// Mitsubishi GX Works2 project: ex2 final   PLC: FX3G
// ex2

// global labels: Global1
VAR_GLOBAL
  start_sys AT X007 : BOOL;
  emergency AT X005 : BOOL;
  led_start AT Y007 : BOOL;
  lack_material AT M0 : BOOL;
  lemon_input AT D1100 : REAL;
  lemon_amount AT D1110 : REAL;
  petel_input AT D1120 : REAL;
  petel_amount AT D1130 : REAL;
  stable_input AT D1140 : REAL;
  stable_amount AT D1150 : REAL;
  bear_input AT D1160 : REAL;
  bear_amount AT D1170 : REAL;
  start_flavor AT X001 : BOOL;
  per_400 AT E400 : REAL;
  pinuk_min AT E6 : REAL;
  pinuk_selected AT M1 : BOOL;
  regular_max AT E5 : REAL;
  regular_selected AT M2 : BOOL;
  lemon_min_pinuk AT E665 : REAL;
  check_lemon_pinuk AT M10 : BOOL;
  check_petel_pinuk AT M30 : BOOL;
  petel_min_pinuk AT E385 : REAL;
  stable_min_pinuk AT E210 : REAL;
  check_stable_pinuk AT M50 : BOOL;
  check_bear_pinuk AT M70 : BOOL;
  bear_min_pinuk AT E70 : REAL;
  can_pinuk AT M3 : BOOL;
  check_lemon_reg AT M11 : BOOL;
  lemon_min_reg AT E455 : REAL;
  check_petel_reg AT M31 : BOOL;
  petel_min_reg AT E280 : REAL;
  check_stable_reg AT M51 : BOOL;
  stable_min_reg AT E105 : REAL;
  bear_min_reg AT E28 : REAL;
  check_bear_reg AT M71 : BOOL;
  can_reg AT M4 : BOOL;
  flavor_timer AT TC1 : BOOL;
  done_flavor AT K50 : INT;
  flavor_mix AT TS1 : BOOL;
  flavor_process AT Y000 : BOOL;
  save_analog_input1 AT D7000 : REAL;
  analog_input1 AT D8280 : INT;
  cooling_done AT M7 : BOOL;
  start_blinking AT M8 : BOOL;
  help_blinker AT M9 : BOOL;
  blinkY5 AT TC2 : BOOL;
  blink_time AT K5 : INT;
  blink1 AT TS2 : BOOL;
  lightY5 AT Y005 : BOOL;
  blinkY6 AT TC3 : BOOL;
  blink2 AT TS3 : BOOL;
  lightY6 AT Y006 : BOOL;
  mix_pinuk AT TS4 : BOOL;
  mix_reg AT TS5 : BOOL;
  done_mix_pinuk AT K50 : INT;
  done_mix_reg AT K30 : INT;
  mix_pinuk_timer AT TC4 : BOOL;
  mix_reg_timer AT TC5 : BOOL;
  pinuk_max AT E10 : REAL;
  regular_min AT E0 : REAL;
  finish_ice_making AT M5 : BOOL;
  start_cool AT X002 : BOOL;
  cool_timer AT TS6 : BOOL;
END_VAR
VAR_GLOBAL CONSTANT
  t_value : INT := 80;
END_VAR
VAR_GLOBAL
  cool_run AT TC6 : BOOL;
  cool_indicator AT Y002 : BOOL;
  finish_cool AT X003 : BOOL;
  start_packege AT X004 : BOOL;
  unit_pack AT X000 : BOOL;
  units_num AT CC1 : BOOL;
END_VAR
VAR_GLOBAL CONSTANT
  const7 : INT := 7;
END_VAR
VAR_GLOBAL
  packege_done AT CS1 : BOOL;
  packege_in_process AT Y004 : BOOL;
  packege_inventory AT D6000 : INT;
END_VAR
VAR_GLOBAL CONSTANT
  const1 : INT := 1;
  const10 : INT := 10;
  K_40 : INT := 40;
END_VAR
VAR_GLOBAL
  analog_output AT D8282 : INT;
  cool_lemon AT D7100 : REAL;
  cool_petel AT D7500 : REAL;
  mix_flavor AT D7400 : REAL;
  mix_with_bear AT D7600 : REAL;
  petel_ice_reg AT E350 : REAL;
  lemon_ice_reg AT E490 : REAL;
  petel_ice_pinuk AT E560 : REAL;
  lemon_ice_pinuk AT E700 : REAL;
END_VAR
VAR_GLOBAL CONSTANT
  bear_reg : REAL := E28;
  bear_pinuk : REAL := E70;
END_VAR
VAR_GLOBAL
  packege_indicator AT M6 : BOOL;
END_VAR

// task Task_01 (event TRUE, interval 0, priority 31): POU_01

PROGRAM POU_01
(* structured ladder/FBD written out as ST: instructions are called as NAME(EN, inputs, outputs); _pN, _eN, _tN stand for wires *)
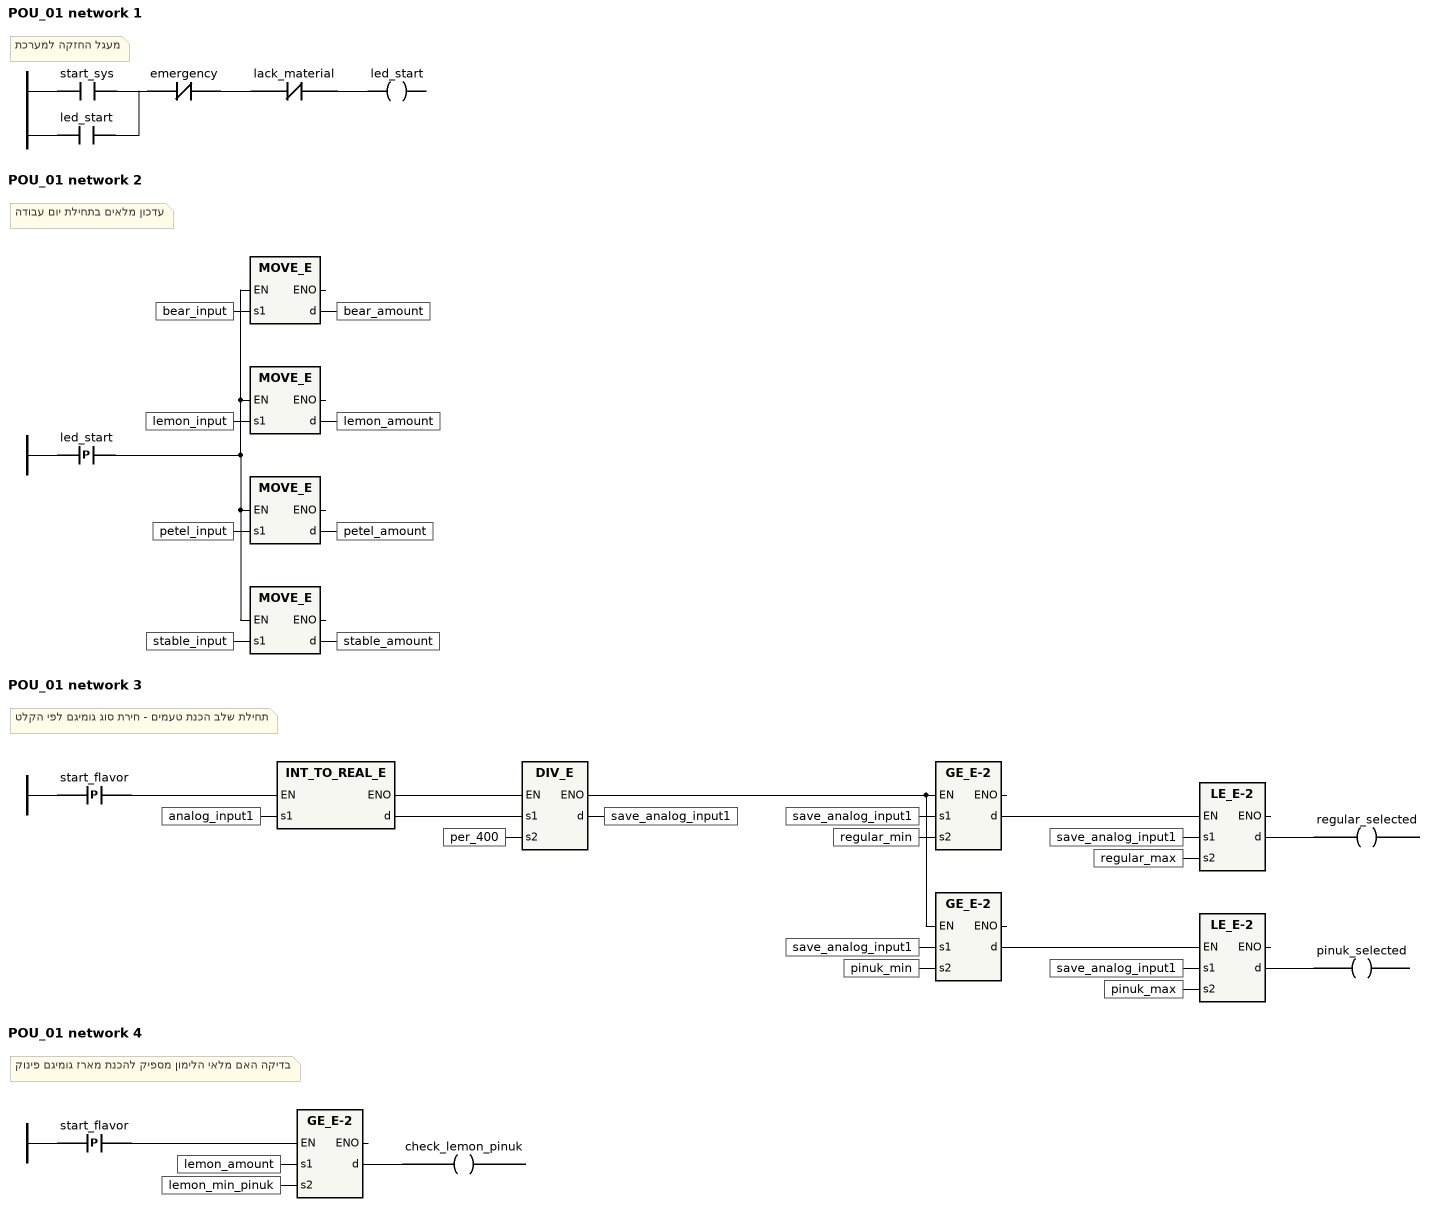
(* network 1 *)
(* מעגל החזקה למערכת *)
led_start := ((start_sys OR led_start) AND NOT emergency) AND NOT lack_material;
(* network 2 *)
(* עדכון מלאים בתחילת יום עבודה *)
_p1 := LDP(TRUE, led_start);
MOVE_E(_p1, bear_input, bear_amount);
MOVE_E(_p1, lemon_input, lemon_amount);
MOVE_E(_p1, petel_input, petel_amount);
MOVE_E(_p1, stable_input, stable_amount);
(* network 3 *)
(* תחילת שלב הכנת טעמים - חירת סוג גומיגם לפי הקלט *)
_e2 := INT_TO_REAL_E(LDP(TRUE, start_flavor), analog_input1, _t1);
_e3 := DIV_E(_e2, _t1, per_400, save_analog_input1);
GE_E(_e3, save_analog_input1, regular_min, _t4);
LE_E(_t4, save_analog_input1, regular_max, _t5);
regular_selected := _t5;
GE_E(_e3, save_analog_input1, pinuk_min, _t6);
LE_E(_t6, save_analog_input1, pinuk_max, _t7);
pinuk_selected := _t7;
(* network 4 *)
(* בדיקה האם מלאי הלימון מספיק להכנת מארז גומיגם פינוק *)
GE_E(LDP(TRUE, start_flavor), lemon_amount, lemon_min_pinuk, _t1);
check_lemon_pinuk := _t1;
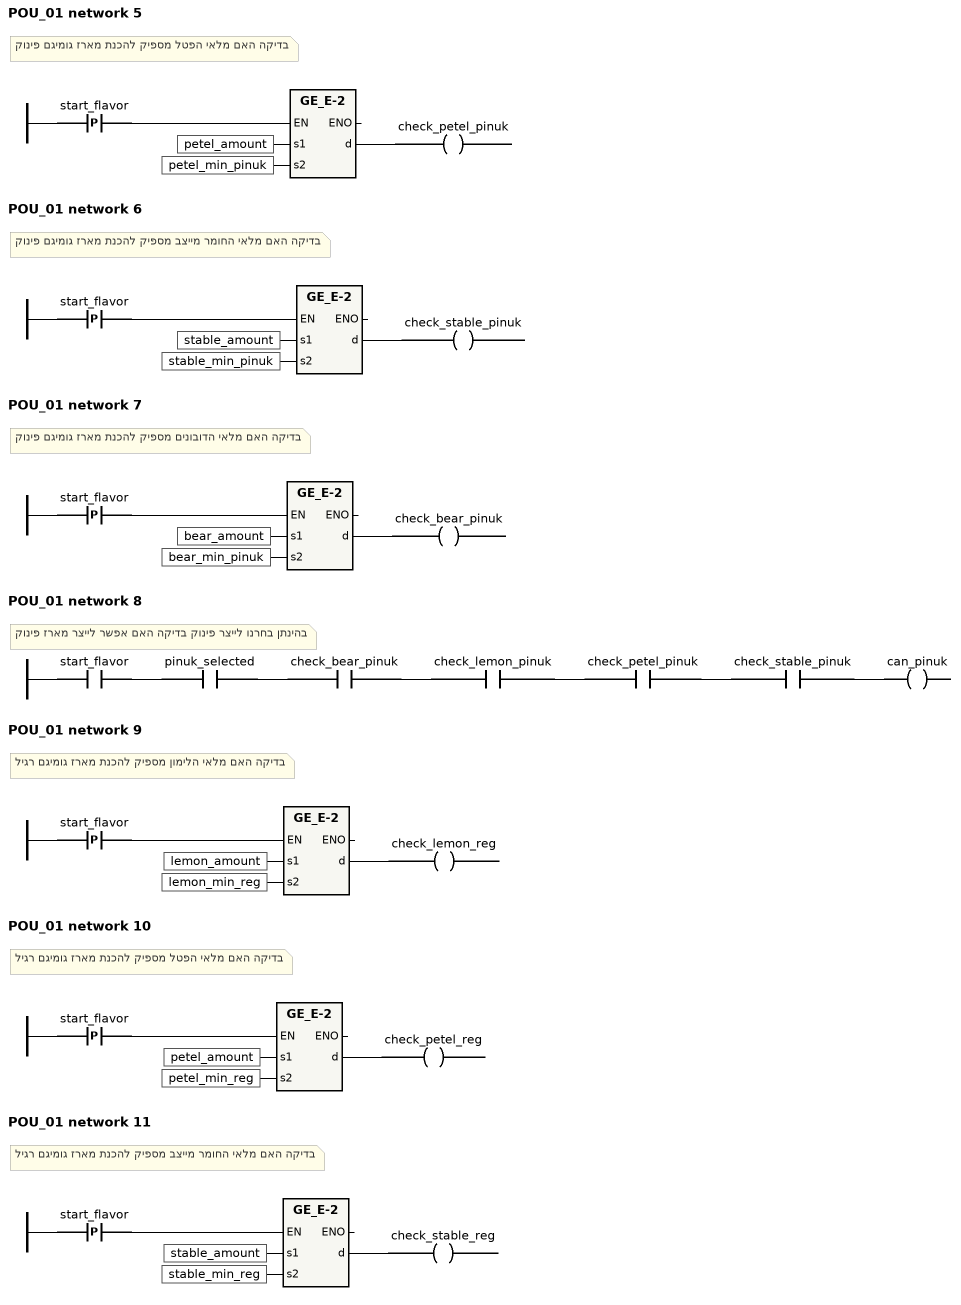
(* network 5 *)
(* בדיקה האם מלאי הפטל מספיק להכנת מארז גומיגם פינוק *)
GE_E(LDP(TRUE, start_flavor), petel_amount, petel_min_pinuk, _t1);
check_petel_pinuk := _t1;
(* network 6 *)
(* בדיקה האם מלאי החומר מייצב מספיק להכנת מארז גומיגם פינוק *)
GE_E(LDP(TRUE, start_flavor), stable_amount, stable_min_pinuk, _t1);
check_stable_pinuk := _t1;
(* network 7 *)
(* בדיקה האם מלאי הדובונים מספיק להכנת מארז גומיגם פינוק *)
GE_E(LDP(TRUE, start_flavor), bear_amount, bear_min_pinuk, _t1);
check_bear_pinuk := _t1;
(* network 8 *)
(* בהינתן בחרנו לייצר פינוק בדיקה האם אפשר לייצר מארז פינוק *)
can_pinuk := start_flavor AND pinuk_selected AND check_bear_pinuk AND check_lemon_pinuk AND check_petel_pinuk AND check_stable_pinuk;
(* network 9 *)
(* בדיקה האם מלאי הלימון מספיק להכנת מארז גומיגם רגיל *)
GE_E(LDP(TRUE, start_flavor), lemon_amount, lemon_min_reg, _t1);
check_lemon_reg := _t1;
(* network 10 *)
(* בדיקה האם מלאי הפטל מספיק להכנת מארז גומיגם רגיל *)
GE_E(LDP(TRUE, start_flavor), petel_amount, petel_min_reg, _t1);
check_petel_reg := _t1;
(* network 11 *)
(* בדיקה האם מלאי החומר מייצב מספיק להכנת מארז גומיגם רגיל *)
GE_E(LDP(TRUE, start_flavor), stable_amount, stable_min_reg, _t1);
check_stable_reg := _t1;
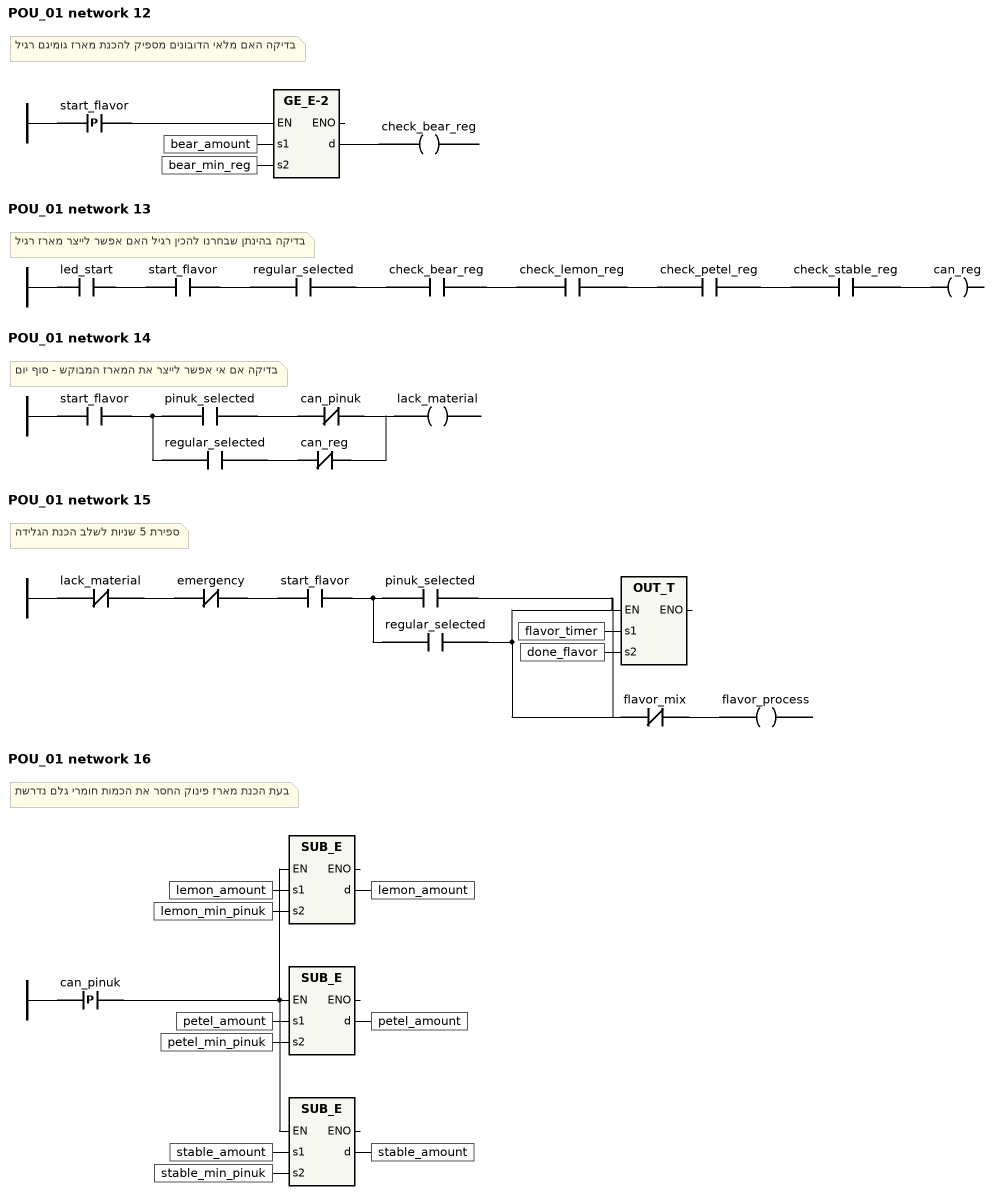
(* network 12 *)
(* בדיקה האם מלאי הדובונים מספיק להכנת מארז גומיגם רגיל *)
GE_E(LDP(TRUE, start_flavor), bear_amount, bear_min_reg, _t1);
check_bear_reg := _t1;
(* network 13 *)
(* בדיקה בהינתן שבחרנו להכין רגיל האם אפשר לייצר מארז רגיל *)
can_reg := led_start AND start_flavor AND regular_selected AND check_bear_reg AND check_lemon_reg AND check_petel_reg AND check_stable_reg;
(* network 14 *)
(* בדיקה אם אי אפשר לייצר את המארז המבוקש - סוף יום *)
lack_material := (start_flavor AND pinuk_selected AND NOT can_pinuk) OR (start_flavor AND regular_selected AND NOT can_reg);
(* network 15 *)
(* ספירת 5 שניות לשלב הכנת הגלידה *)
_p1 := NOT lack_material AND NOT emergency AND start_flavor;
_p2 := (_p1 AND pinuk_selected) OR (_p1 AND regular_selected);
flavor_process := _p2 AND NOT flavor_mix;
OUT_T(_p2, flavor_timer, done_flavor);
(* network 16 *)
(* בעת הכנת מארז פינוק החסר את הכמות חומרי גלם נדרשת *)
_p1 := LDP(TRUE, can_pinuk);
SUB_E(_p1, lemon_amount, lemon_min_pinuk, lemon_amount);
SUB_E(_p1, petel_amount, petel_min_pinuk, petel_amount);
SUB_E(_p1, stable_amount, stable_min_pinuk, stable_amount);
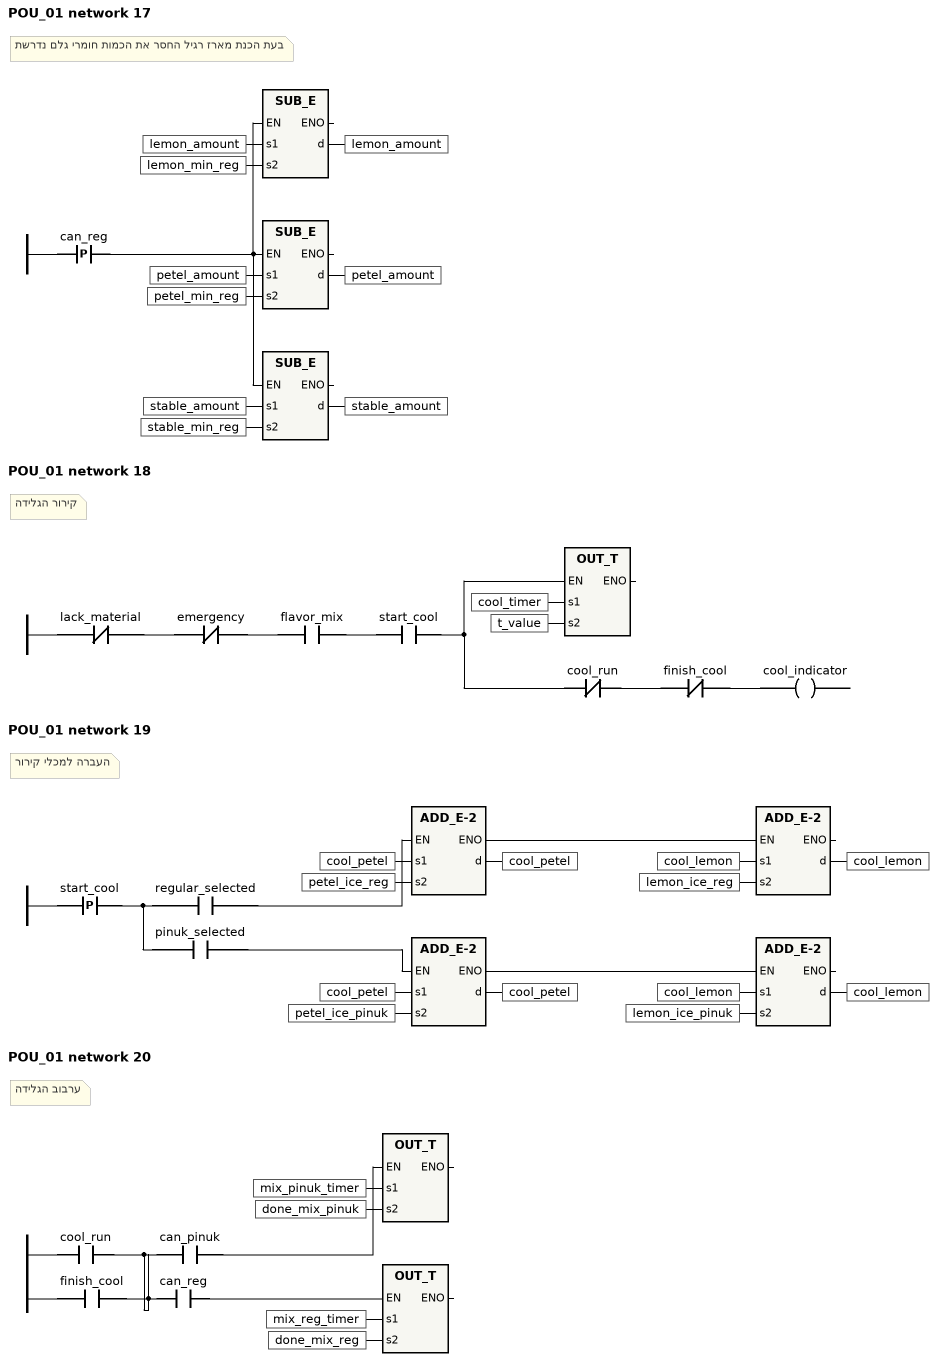
(* network 17 *)
(* בעת הכנת מארז רגיל החסר את הכמות חומרי גלם נדרשת *)
_p1 := LDP(TRUE, can_reg);
SUB_E(_p1, lemon_amount, lemon_min_reg, lemon_amount);
SUB_E(_p1, petel_amount, petel_min_reg, petel_amount);
SUB_E(_p1, stable_amount, stable_min_reg, stable_amount);
(* network 18 *)
(* קירור הגלידה *)
_p1 := NOT lack_material AND NOT emergency AND flavor_mix AND start_cool;
OUT_T(_p1, cool_timer, t_value);
cool_indicator := _p1 AND NOT cool_run AND NOT finish_cool;
(* network 19 *)
(* העברה למכלי קירור *)
_p1 := LDP(TRUE, start_cool);
_e2 := ADD_E(_p1 AND regular_selected, cool_petel, petel_ice_reg, cool_petel);
ADD_E(_e2, cool_lemon, lemon_ice_reg, cool_lemon);
_e3 := ADD_E(_p1 AND pinuk_selected, cool_petel, petel_ice_pinuk, cool_petel);
ADD_E(_e3, cool_lemon, lemon_ice_pinuk, cool_lemon);
(* network 20 *)
(* ערבוב הגלידה *)
_p1 := cool_run OR finish_cool;
OUT_T(_p1 AND can_pinuk, mix_pinuk_timer, done_mix_pinuk);
OUT_T(_p1 AND can_reg, mix_reg_timer, done_mix_reg);
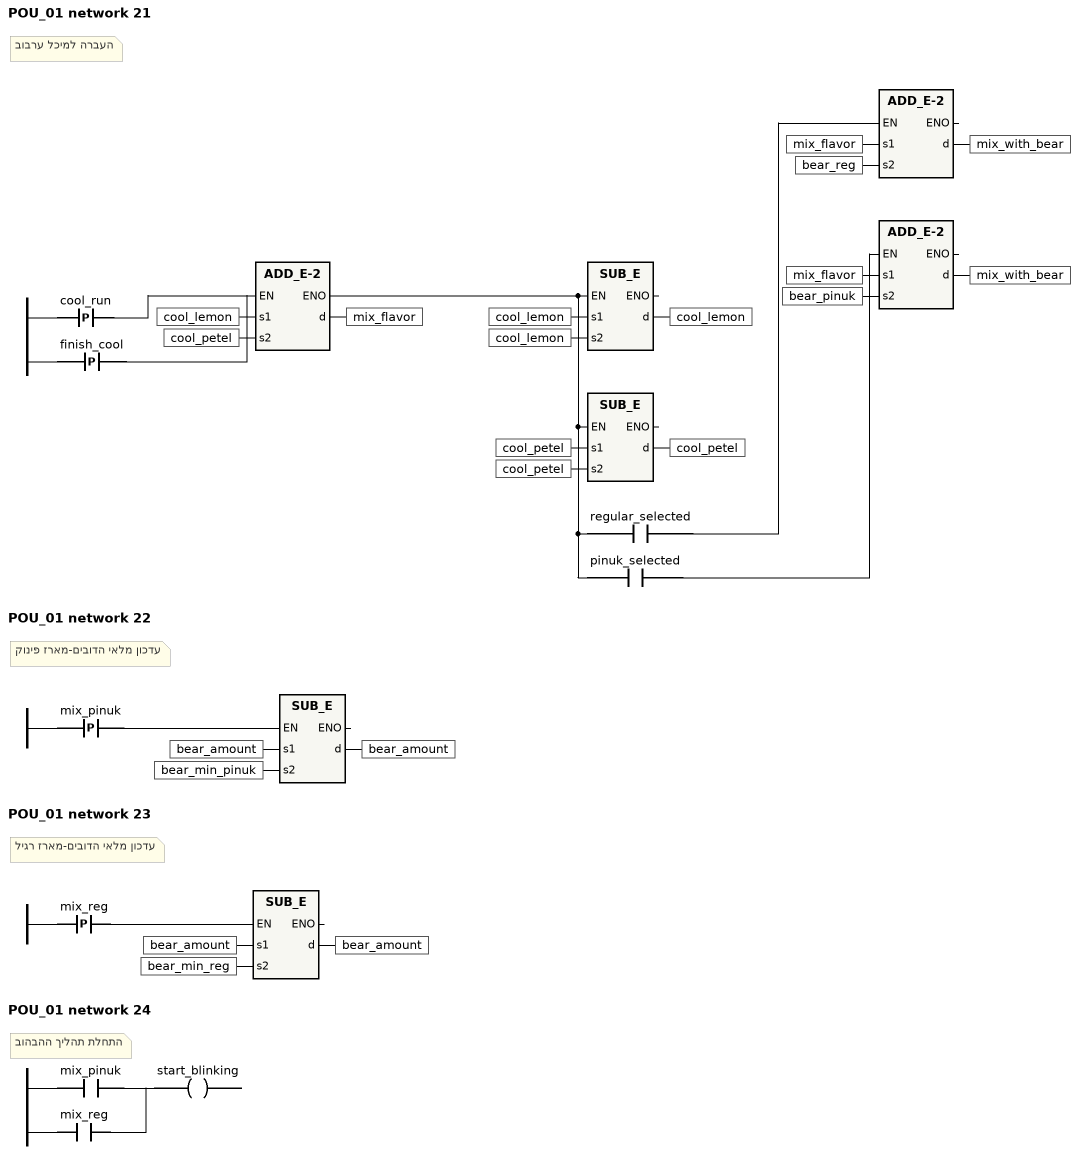
(* network 21 *)
(* העברה למיכל ערבוב *)
_e1 := ADD_E(LDP(TRUE, cool_run) OR LDP(TRUE, finish_cool), cool_lemon, cool_petel, mix_flavor);
ADD_E(_e1 AND regular_selected, mix_flavor, bear_reg, mix_with_bear);
ADD_E(_e1 AND pinuk_selected, mix_flavor, bear_pinuk, mix_with_bear);
SUB_E(_e1, cool_lemon, cool_lemon, cool_lemon);
SUB_E(_e1, cool_petel, cool_petel, cool_petel);
(* network 22 *)
(* עדכון מלאי הדובים-מארז פינוק *)
SUB_E(LDP(TRUE, mix_pinuk), bear_amount, bear_min_pinuk, bear_amount);
(* network 23 *)
(* עדכון מלאי הדובים-מארז רגיל *)
SUB_E(LDP(TRUE, mix_reg), bear_amount, bear_min_reg, bear_amount);
(* network 24 *)
(* התחלת תהליך ההבהוב *)
start_blinking := mix_pinuk OR mix_reg;
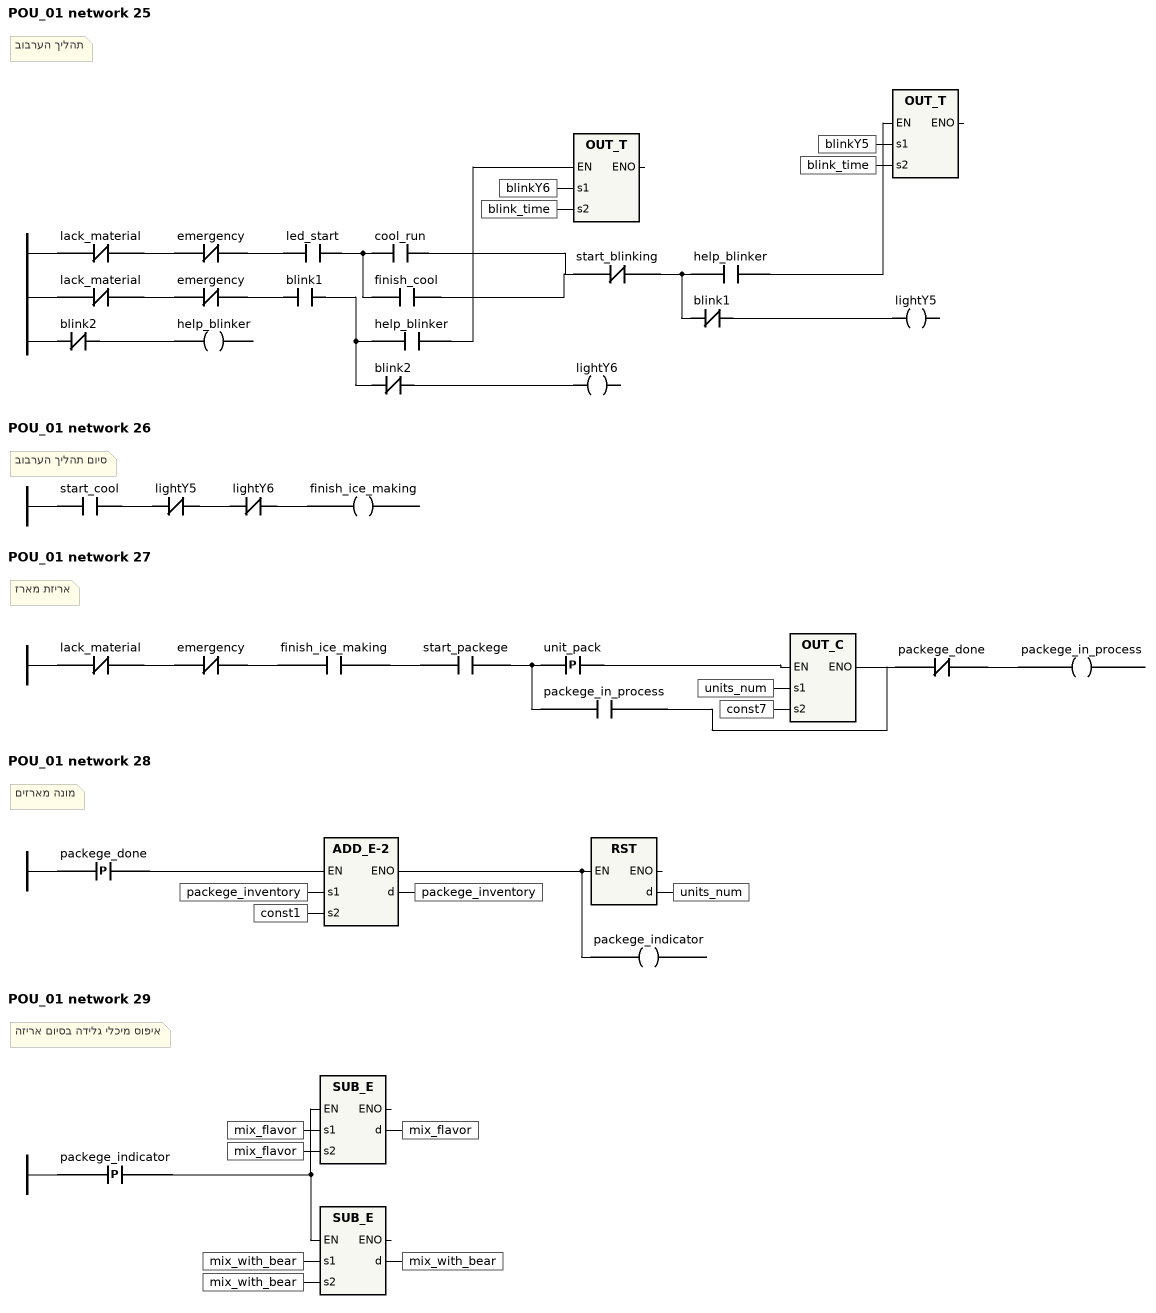
(* network 25 *)
(* תהליך הערבוב *)
_p1 := NOT lack_material AND NOT emergency AND led_start;
_p2 := ((_p1 AND cool_run) OR (_p1 AND finish_cool)) AND NOT start_blinking;
OUT_T(_p2 AND help_blinker, blinkY5, blink_time);
lightY5 := _p2 AND NOT blink1;
_p3 := NOT lack_material AND NOT emergency AND blink1;
OUT_T(_p3 AND help_blinker, blinkY6, blink_time);
lightY6 := _p3 AND NOT blink2;
help_blinker := NOT blink2;
(* network 26 *)
(* סיום תהליך הערבוב *)
finish_ice_making := start_cool AND NOT lightY5 AND NOT lightY6;
(* network 27 *)
(* אריזת מארז *)
_p1 := NOT lack_material AND NOT emergency AND finish_ice_making AND start_packege;
_e2 := OUT_C(_p1 AND LDP(TRUE, unit_pack), units_num, const7);
packege_in_process := (_e2 OR (_p1 AND packege_in_process)) AND NOT packege_done;
(* network 28 *)
(* מונה מארזים *)
_e1 := ADD_E(LDP(TRUE, packege_done), packege_inventory, const1, packege_inventory);
packege_indicator := _e1;
RST(_e1, units_num);
(* network 29 *)
(* איפוס מיכלי גלידה בסיום אריזה *)
_p1 := LDP(TRUE, packege_indicator);
SUB_E(_p1, mix_flavor, mix_flavor, mix_flavor);
SUB_E(_p1, mix_with_bear, mix_with_bear, mix_with_bear);
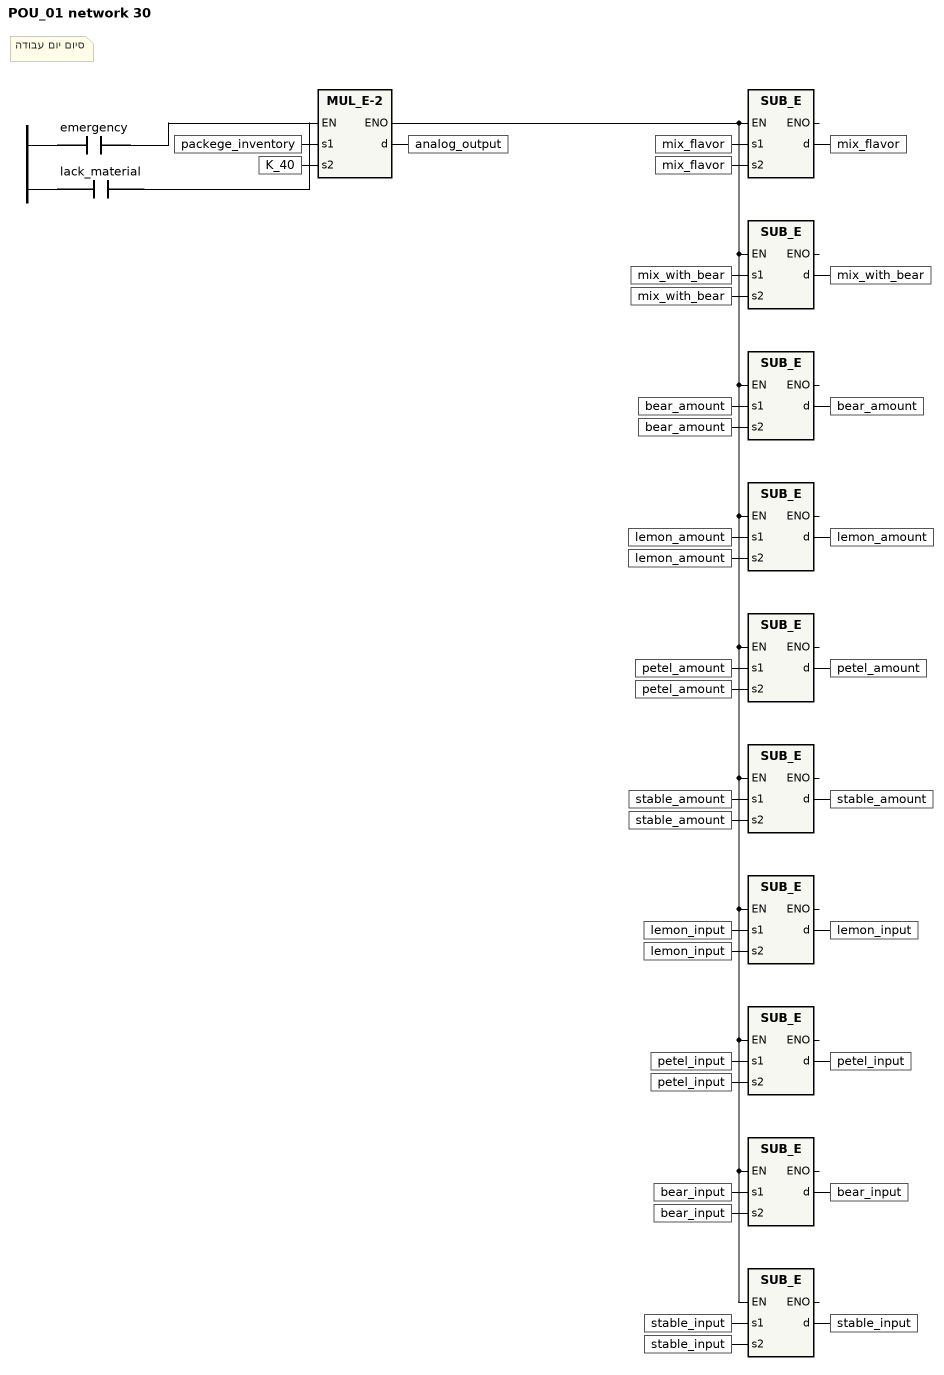
(* network 30 *)
(* סיום יום עבודה *)
_e1 := MUL_E(emergency OR lack_material, packege_inventory, K_40, analog_output);
SUB_E(_e1, mix_flavor, mix_flavor, mix_flavor);
SUB_E(_e1, mix_with_bear, mix_with_bear, mix_with_bear);
SUB_E(_e1, bear_amount, bear_amount, bear_amount);
SUB_E(_e1, lemon_amount, lemon_amount, lemon_amount);
SUB_E(_e1, petel_amount, petel_amount, petel_amount);
SUB_E(_e1, stable_amount, stable_amount, stable_amount);
SUB_E(_e1, lemon_input, lemon_input, lemon_input);
SUB_E(_e1, petel_input, petel_input, petel_input);
SUB_E(_e1, bear_input, bear_input, bear_input);
SUB_E(_e1, stable_input, stable_input, stable_input);
END_PROGRAM
